// TIA Portal project "Fechamento" (V17)

(* hardware
DEVICE "S7-300/ET200M station_1"  S7-300 station
   slot 0: "Rail_0"  Rail  6ES7 390-1***0-0AA0
   slot 2: "PLC_1"  CPU 319F-3 PN/DP  6ES7 318-3FL01-0AB0  V3.2
      slot 2: "DP interface_1"  DP
      slot 3: "PROFINET interface_1"  PN-IO
         slot 1: "Port_1"  Port
         slot 2: "Port_2"  Port
*)

// ===== PLC "PLC_1"  CPU 319F-3 PN/DP =====

VAR_GLOBAL   // PLC tag table "Default tag table"
   "Esteira" AT %Q0.0 : Bool;
   "Botão_Liga_Esteira" AT %I0.0 : Bool;
   "Sensor_Posição" AT %I0.1 : Bool;
   "Pistão_1" AT %Q0.1 : Bool;
   "Pistão_2" AT %Q0.2 : Bool;
   "Pistão_Prensa" AT %Q0.3 : Bool;
   "Sensor_Prensa_Recuado" AT %I0.2 : Bool;
   "Sensor_Prensa_Avançado" AT %I0.3 : Bool;
   "Motor_Vácuo_Tampa" AT %Q0.4 : Bool;
   "Sensor_Reserva_Tampa" AT %I0.4 : Bool;
   "Lampada_Reserva_Tampa" AT %Q0.5 : Bool;
   "Botão_Desliga" AT %I0.5 : Bool;
   "Botão_Emergência" AT %I0.6 : Bool;
   "Lampada_Emergência" AT %Q0.6 : Bool;
   "Desliga_Pistão_2" AT %Q0.7 : Bool;
   "Tag_1" AT %M0.0 : Bool;
   "Tag_2" AT %M0.1 : Bool;
END_VAR

FUNCTION "Block_1" : Void   // FC1, LAD
{ S7_Optimized_Access := 'FALSE' }
VERSION : 0.1
BEGIN

REGION Network 1
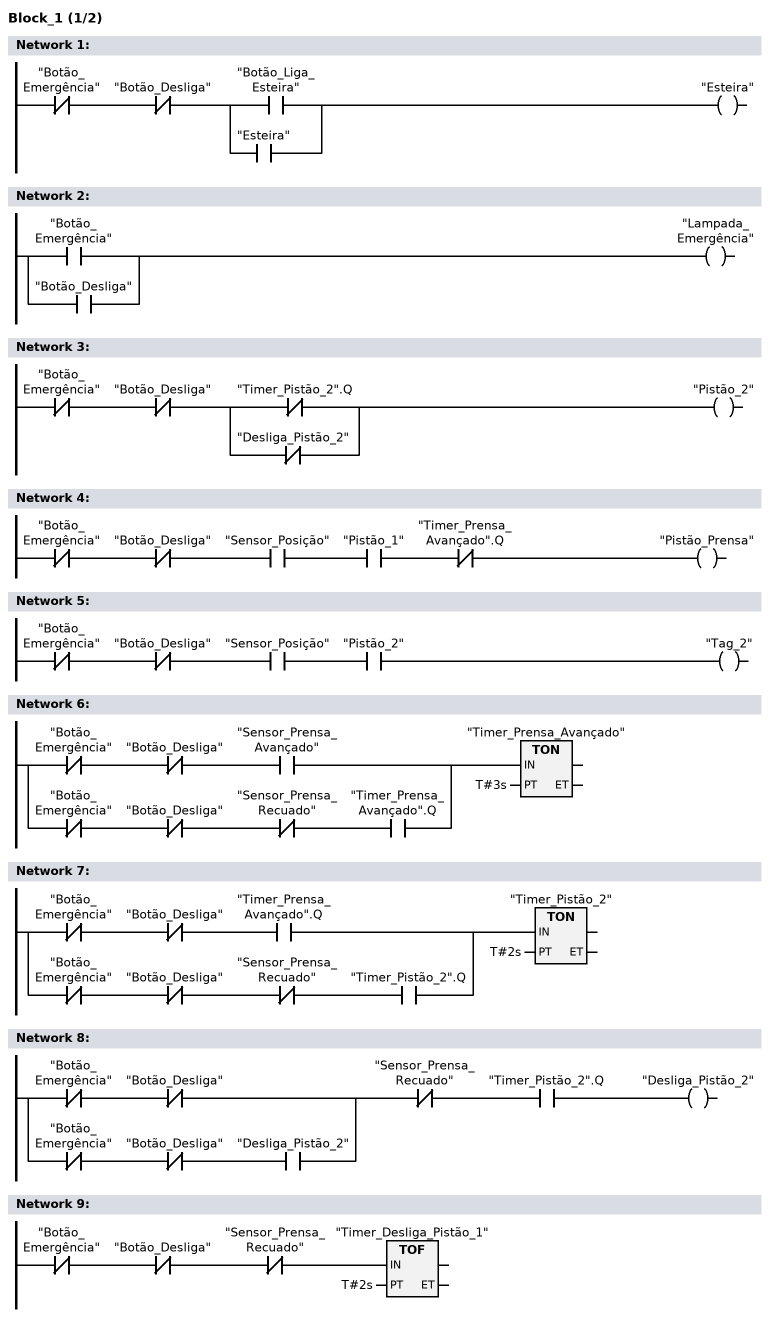
   RUNG wire#powerrail
      I_Contact( "Botão_Emergência" )
      I_Contact( "Botão_Desliga" )
      wire#w1
      Contact( "Botão_Liga_Esteira" )
      wire#w2
      Coil( "Esteira" )
   END_RUNG
   RUNG wire#w1
      Contact( "Esteira" )
   END_RUNG wire#w2
   // the same network as SCL:
   "Esteira" := NOT "Botão_Emergência" AND NOT "Botão_Desliga" AND ("Botão_Liga_Esteira" OR "Esteira");
END_REGION

REGION Network 2
   RUNG wire#powerrail
      Contact( "Botão_Emergência" )
      wire#w1
      Coil( "Lampada_Emergência" )
   END_RUNG
   RUNG wire#powerrail
      Contact( "Botão_Desliga" )
   END_RUNG wire#w1
   // the same network as SCL:
   "Lampada_Emergência" := "Botão_Emergência" OR "Botão_Desliga";
END_REGION

REGION Network 3
   RUNG wire#powerrail
      I_Contact( "Botão_Emergência" )
      I_Contact( "Botão_Desliga" )
      wire#w1
      I_Contact( "Timer_Pistão_2".Q )
      wire#w2
      Coil( "Pistão_2" )
   END_RUNG
   RUNG wire#w1
      I_Contact( "Desliga_Pistão_2" )
   END_RUNG wire#w2
   // the same network as SCL:
   "Pistão_2" := NOT "Botão_Emergência" AND NOT "Botão_Desliga" AND (NOT "Timer_Pistão_2".Q OR NOT "Desliga_Pistão_2");
END_REGION

REGION Network 4
   RUNG wire#powerrail
      I_Contact( "Botão_Emergência" )
      I_Contact( "Botão_Desliga" )
      Contact( "Sensor_Posição" )
      Contact( "Pistão_1" )
      I_Contact( "Timer_Prensa_Avançado".Q )
      Coil( "Pistão_Prensa" )
   END_RUNG
   // the same network as SCL:
   "Pistão_Prensa" := NOT "Botão_Emergência" AND NOT "Botão_Desliga" AND "Sensor_Posição" AND "Pistão_1" AND NOT "Timer_Prensa_Avançado".Q;
END_REGION

REGION Network 5
   RUNG wire#powerrail
      I_Contact( "Botão_Emergência" )
      I_Contact( "Botão_Desliga" )
      Contact( "Sensor_Posição" )
      Contact( "Pistão_2" )
      Coil( "Tag_2" )
   END_RUNG
   // the same network as SCL:
   "Tag_2" := NOT "Botão_Emergência" AND NOT "Botão_Desliga" AND "Sensor_Posição" AND "Pistão_2";
END_REGION

REGION Network 6
   "Timer_Prensa_Avançado".TON(IN := (NOT "Botão_Emergência" AND NOT "Botão_Desliga" AND "Sensor_Prensa_Avançado") OR (NOT "Botão_Emergência" AND NOT "Botão_Desliga" AND NOT "Sensor_Prensa_Recuado" AND "Timer_Prensa_Avançado".Q),
                           PT := T#3s);
END_REGION

REGION Network 7
   "Timer_Pistão_2".TON(IN := (NOT "Botão_Emergência" AND NOT "Botão_Desliga" AND "Timer_Prensa_Avançado".Q) OR (NOT "Botão_Emergência" AND NOT "Botão_Desliga" AND NOT "Sensor_Prensa_Recuado" AND "Timer_Pistão_2".Q),
                        PT := T#2s);
END_REGION

REGION Network 8
   RUNG wire#powerrail
      I_Contact( "Botão_Emergência" )
      I_Contact( "Botão_Desliga" )
      wire#w1
      I_Contact( "Sensor_Prensa_Recuado" )
      Contact( "Timer_Pistão_2".Q )
      Coil( "Desliga_Pistão_2" )
   END_RUNG
   RUNG wire#powerrail
      I_Contact( "Botão_Emergência" )
      I_Contact( "Botão_Desliga" )
      Contact( "Desliga_Pistão_2" )
   END_RUNG wire#w1
   // the same network as SCL:
   "Desliga_Pistão_2" := ((NOT "Botão_Emergência" AND NOT "Botão_Desliga") OR (NOT "Botão_Emergência" AND NOT "Botão_Desliga" AND "Desliga_Pistão_2")) AND NOT "Sensor_Prensa_Recuado" AND "Timer_Pistão_2".Q;
END_REGION

REGION Network 9
   "Timer_Desliga_Pistão_1".TOF(IN := NOT "Botão_Emergência" AND NOT "Botão_Desliga" AND NOT "Sensor_Prensa_Recuado",
                           PT := T#2s);
END_REGION

REGION Network 10
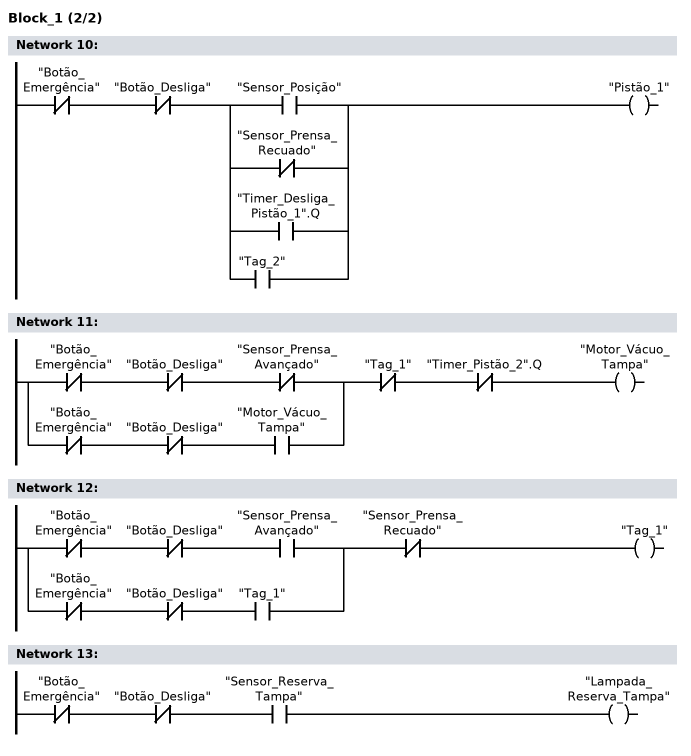
   RUNG wire#powerrail
      I_Contact( "Botão_Emergência" )
      I_Contact( "Botão_Desliga" )
      wire#w1
      Contact( "Sensor_Posição" )
      wire#w2
      Coil( "Pistão_1" )
   END_RUNG
   RUNG wire#w1
      I_Contact( "Sensor_Prensa_Recuado" )
   END_RUNG wire#w2
   RUNG wire#w1
      Contact( "Timer_Desliga_Pistão_1".Q )
   END_RUNG wire#w2
   RUNG wire#w1
      Contact( "Tag_2" )
   END_RUNG wire#w2
   // the same network as SCL:
   "Pistão_1" := NOT "Botão_Emergência" AND NOT "Botão_Desliga" AND ("Sensor_Posição" OR NOT "Sensor_Prensa_Recuado" OR "Timer_Desliga_Pistão_1".Q OR "Tag_2");
END_REGION

REGION Network 11
   RUNG wire#powerrail
      I_Contact( "Botão_Emergência" )
      I_Contact( "Botão_Desliga" )
      I_Contact( "Sensor_Prensa_Avançado" )
      wire#w1
      I_Contact( "Tag_1" )
      I_Contact( "Timer_Pistão_2".Q )
      Coil( "Motor_Vácuo_Tampa" )
   END_RUNG
   RUNG wire#powerrail
      I_Contact( "Botão_Emergência" )
      I_Contact( "Botão_Desliga" )
      Contact( "Motor_Vácuo_Tampa" )
   END_RUNG wire#w1
   // the same network as SCL:
   "Motor_Vácuo_Tampa" := ((NOT "Botão_Emergência" AND NOT "Botão_Desliga" AND NOT "Sensor_Prensa_Avançado") OR (NOT "Botão_Emergência" AND NOT "Botão_Desliga" AND "Motor_Vácuo_Tampa")) AND NOT "Tag_1" AND NOT "Timer_Pistão_2".Q;
END_REGION

REGION Network 12
   RUNG wire#powerrail
      I_Contact( "Botão_Emergência" )
      I_Contact( "Botão_Desliga" )
      Contact( "Sensor_Prensa_Avançado" )
      wire#w1
      I_Contact( "Sensor_Prensa_Recuado" )
      Coil( "Tag_1" )
   END_RUNG
   RUNG wire#powerrail
      I_Contact( "Botão_Emergência" )
      I_Contact( "Botão_Desliga" )
      Contact( "Tag_1" )
   END_RUNG wire#w1
   // the same network as SCL:
   "Tag_1" := ((NOT "Botão_Emergência" AND NOT "Botão_Desliga" AND "Sensor_Prensa_Avançado") OR (NOT "Botão_Emergência" AND NOT "Botão_Desliga" AND "Tag_1")) AND NOT "Sensor_Prensa_Recuado";
END_REGION

REGION Network 13
   RUNG wire#powerrail
      I_Contact( "Botão_Emergência" )
      I_Contact( "Botão_Desliga" )
      Contact( "Sensor_Reserva_Tampa" )
      Coil( "Lampada_Reserva_Tampa" )
   END_RUNG
   // the same network as SCL:
   "Lampada_Reserva_Tampa" := NOT "Botão_Emergência" AND NOT "Botão_Desliga" AND "Sensor_Reserva_Tampa";
END_REGION
END_FUNCTION

ORGANIZATION_BLOCK "Main"   // OB1, LAD
TITLE = "Main Program Sweep (Cycle)"
{ S7_Optimized_Access := 'FALSE' }
VERSION : 0.1
   VAR_TEMP
      OB1_EV_CLASS : Byte;   // Bits 0-3 = 1 (Coming event), Bits 4-7 = 1 (Event class 1)
      OB1_SCAN_1 : Byte;   // 1 (Cold restart scan 1 of OB 1), 3 (Scan 2-n of OB 1)
      OB1_PRIORITY : Byte;   // Priority of OB Execution
      OB1_OB_NUMBR : Byte;   // 1 (Organization block 1, OB1)
      OB1_RESERVED_1 : Byte;   // Reserved for system
      OB1_RESERVED_2 : Byte;   // Reserved for system
      OB1_PREV_CYCLE : Int;   // Cycle time of previous OB1 scan (milliseconds)
      OB1_MIN_CYCLE : Int;   // Minimum cycle time of OB1 (milliseconds)
      OB1_MAX_CYCLE : Int;   // Maximum cycle time of OB1 (milliseconds)
      OB1_DATE_TIME : Date_And_Time;   // Date and time OB1 started
   END_VAR
BEGIN

REGION Network 1
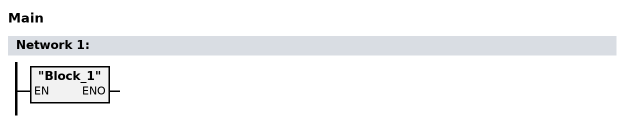
   RUNG wire#powerrail
      "Block_1"()
   END_RUNG
   // the same network as SCL:
   "Block_1"();
END_REGION
END_ORGANIZATION_BLOCK